{attribute 'no_check'}
(* 
输出功能块 Output
输出功能块
*)
FUNCTION_BLOCK Output
VAR_INPUT
	Enable : BOOL := TRUE; (* False: 不启用, True: 启用 *)
END_VAR
VAR_OUTPUT
	Out AT%Q* : BOOL; (* 绑定到输出变量，或者利用功能块引脚直接输出 *)
END_VAR
VAR
	InternCycleCounter : UDINT; (* 执行时内置的循环数 *)
	ThisCycleExecuteCounter : UDINT; (* 当前周期循环数 *)
	LastCycleExecuteCounter : UDINT; (* 上个周期循环数 *)
END_VAR

(*
TIME		: 2023-11-13 15:46
Version		: 1.0
Creator		: Ulysses
Reference	: IOTA - BLUE
Commecnts	: 输出功能块，Set返回值代表当前周期调用次数，LastCounter代表上个周期调用次数。
*)

(* 上周期调用次数 *)
PROPERTY LastCounter : UDINT
GET
LastCounter := LastCycleExecuteCounter;
END_GET
END_PROPERTY

(* 返回值代表当前周期内SetOn或者SetOff被执行的次数，正常为1，如果大于1则可能出现双线圈问题 *)
METHOD SetOff : UDINT
VAR_INPUT
END_VAR
VAR
	TempCycleCounter : UDINT;
END_VAR
Out := Enable AND FALSE;
TempCycleCounter := _TaskInfo[GETCURTASKINDEXEX()].CycleCount;
IF InternCycleCounter <> TempCycleCounter THEN
	InternCycleCounter := TempCycleCounter;
	LastCycleExecuteCounter := ThisCycleExecuteCounter;
	ThisCycleExecuteCounter := 0 ;
END_IF
ThisCycleExecuteCounter := ThisCycleExecuteCounter + 1;

SetOff := ThisCycleExecuteCounter;
END_METHOD

(* 返回值代表当前周期内SetOn或者SetOff被执行的次数，正常为1，如果大于1则可能出现双线圈问题 *)
METHOD SetOn : UDINT
VAR_INPUT
END_VAR
VAR
	TempCycleCounter : UDINT;
END_VAR
Out := Enable AND TRUE;
TempCycleCounter := _TaskInfo[GETCURTASKINDEXEX()].CycleCount;
IF InternCycleCounter <> TempCycleCounter THEN
	InternCycleCounter := TempCycleCounter;
	LastCycleExecuteCounter := ThisCycleExecuteCounter;
	ThisCycleExecuteCounter := 0 ;
END_IF
ThisCycleExecuteCounter := ThisCycleExecuteCounter + 1;

SetOn := ThisCycleExecuteCounter;
END_METHOD

END_FUNCTION_BLOCK

(* stored: Version 1.1.0.1, ProductVersion 3.1.4024.12
   POU Output: Id {472376e7-6ad9-48cc-93bb-cc7e5b404f58}, SpecialFunc None
   Property LastCounter: Id {a1899f5b-4114-4790-b81c-0aac29c23635}
   Get Get: Id {8eb5f064-9d3f-4304-bd34-3c3b56577024}
   Method SetOff: Id {c2d2f019-cd2d-42f1-92b5-573c526d4460}
   Method SetOn: Id {99401f8e-b942-43b3-a676-ffa1da7caa66} *)
